DATA_BLOCK "DB_BOX_1"
{ S7_Optimized_Access := 'TRUE' }
VERSION : 0.1
NON_RETAIN
"FB_easyBox"

BEGIN

END_DATA_BLOCK

